FUNCTION_BLOCK FB_EpicsInOut_Test EXTENDS TcUnit.FB_TestSuite
VAR
    Expected: BOOL;
    Actual: BOOL;
END_VAR

TEST('FB_EpicsInOut_Test Dummy Test');
AssertEquals(Expected := Expected,
             Actual := Actual,
             Message := 'Error Message');
TEST_FINISHED();

END_FUNCTION_BLOCK

(* stored: Version 1.1.0.1, ProductVersion 3.1.4022.18
   POU FB_EpicsInOut_Test: Id {eef9e40b-2155-4b64-be43-4e763da61f99}, SpecialFunc None *)
